// TwinCAT 3 PLC project Sample01
// ProgramVersion: 3.1.4022.4
// libraries:
//   Tc2_Standard, * (Beckhoff Automation GmbH)
//   Tc2_System, * (Beckhoff Automation GmbH)
//   Tc3_Module, * (Beckhoff Automation GmbH)
// project tree:
//   / ClassDiagram.TcCD (not stored), PlcTask.TcTTO
//   DUTs/ E_PizzaStyle.TcDUT
//   POUs/ FB_Pizza.TcPOU, MAIN.TcPOU
// real-time tasks:
//   TASK PlcTask: cycle T#10ms, priority 20, ADS port 350

CONFIGURATION Sample01
    RESOURCE PLC ON TwinCAT3
        TASK PlcTask(INTERVAL := T#10ms, PRIORITY := 20);
        PROGRAM MAIN WITH PlcTask : MAIN;
    END_RESOURCE
END_CONFIGURATION

// ---- DUTs/E_PizzaStyle.TcDUT
{attribute 'qualified_only'}
{attribute 'strict'}
TYPE E_PizzaStyle :
(
	eAmerican	:= 0,
	eItalian	:= 1
);
END_TYPE

// ---- POUs/MAIN.TcPOU
PROGRAM MAIN
VAR
	fbAmericanSalamiPizza		: FB_Pizza(ePizzaStyle := E_PizzaStyle.eAmerican, bHasBroccoli := FALSE, bHasCheese := TRUE, bHasSalami := TRUE);
	fbItalianVegetarianPizza	: FB_Pizza(ePizzaStyle := E_PizzaStyle.eItalian, bHasBroccoli := TRUE, bHasCheese := FALSE, bHasSalami := FALSE);
END_VAR

END_PROGRAM

// ---- POUs/FB_Pizza.TcPOU
FUNCTION_BLOCK PUBLIC FB_Pizza
VAR_INPUT
END_VAR
VAR_OUTPUT
END_VAR
VAR
	eStyle		: E_PizzaStyle;
	bBroccoli	: BOOL;
	bCheese		: BOOL;
	bSalami		: BOOL;
END_VAR

PROPERTY PUBLIC bHasBroccoli : BOOL
GET
bHasBroccoli := this^.bBroccoli;
END_GET
SET
this^.bBroccoli := bHasBroccoli;
END_SET
END_PROPERTY

PROPERTY PUBLIC bHasCheese : BOOL
GET
bHasCheese := this^.bCheese;
END_GET
SET
this^.bCheese := bHasCheese;
END_SET
END_PROPERTY

PROPERTY PUBLIC bHasSalami : BOOL
GET
bHasSalami := this^.bSalami;
END_GET
SET
this^.bSalami := bHasSalami;
END_SET
END_PROPERTY

PROPERTY PUBLIC ePizzaStyle : E_PizzaStyle
GET
ePizzaStyle := this^.eStyle;
END_GET
SET
this^.eStyle := ePizzaStyle;
END_SET
END_PROPERTY

METHOD FB_init : BOOL
VAR_INPUT
	bInitRetains	: BOOL; // if TRUE, the retain variables are initialized (warm start / cold start)
	bInCopyCode		: BOOL;  // if TRUE, the instance afterwards gets moved into the copy code (online change)
	ePizzaStyle		: E_PizzaStyle;
	bHasBroccoli	: BOOL;
	bHasCheese 		: BOOL;
	bHasSalami		: BOOL;
END_VAR
THIS^.eStyle := ePizzaStyle;
THIS^.bBroccoli := bHasBroccoli;
THIS^.bCheese := bHasCheese;
this^.bSalami := bHasSalami;
END_METHOD

METHOD PUBLIC GetPrice : LREAL
IF (THIS^.eStyle = E_PizzaStyle.eItalian) THEN
	GetPrice := 4.5;
ELSIF (THIS^.eStyle = E_PizzaStyle.eAmerican) THEN
	GetPrice := 4.2;
ELSE
	GetPrice := 0;
	RETURN;
END_IF
IF (THIS^.bBroccoli) THEN
	GetPrice := GetPrice + 0.8;
END_IF
IF (THIS^.bCheese) THEN
	GetPrice := GetPrice + 1.1;
END_IF
IF (THIS^.bSalami) THEN
	GetPrice := GetPrice + 1.4;
END_IF
END_METHOD

END_FUNCTION_BLOCK
